Fanuc KAREL source: kb00180.KL

-- PROVISIONAL review KL for V1013-1; original PC SHA256 13ea58bf92d87e1c0af7fb51ab888464c06f0ad45a98962b692b2511957ddb51
-- Incomplete behavior may be omitted. Consult companion uncertainty JSON. Do not deploy.
PROGRAM KB00180
%NOLOCKGROUP
BEGIN
  -- UNRESOLVED_PC offsets 5-12; opcodes 9D,23
  -- UNRESOLVED_PC offsets 17-26; opcodes 3F,75
  -- UNRESOLVED_PC offsets 31-38; opcodes 9D,23
  -- UNRESOLVED_PC offsets 43-67; opcodes 27,22,22,2A,22,31
  -- UNRESOLVED_PC offsets 72-76; opcodes 7F
END KB00180
